// Mitsubishi GX Works2 project: 자기유지   PLC: Q02/Q02H

PROGRAM MAIN
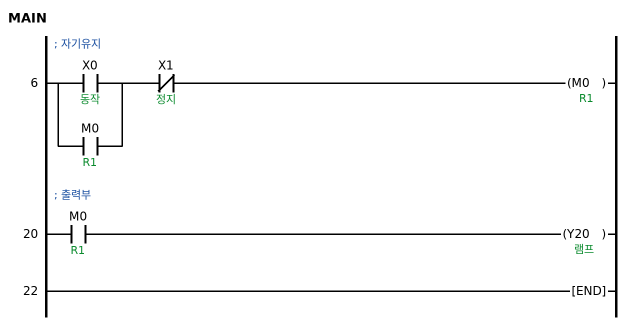
; 자기유지
6     LD      X0  ; 동작
      OR      M0  ; R1
      ANI     X1  ; 정지
      OUT     M0  ; R1
        [note] 릴레이
; 출력부
20    LD      M0  ; R1
      OUT     Y20  ; 램프
22    END
END_PROGRAM
